VISUALIZATION VISU_M1Figure_Valve  // 22x12
    Polygon (0,10) (0,0) (10,5)
    Polygon (20,10) (10,5) (20,0)
END_VISUALIZATION

(* stored: Version 1.1.0.1, ProductVersion 3.1.4018.2
   Visu VISU_M1Figure_Valve: Id {84eba547-86e9-4672-a5b7-7511b6602c05} *)
